PROGRAM PRG_03_Saw
VAR
	b_SRout: BOOL;	
	SR_saw: SR;
	R_TRIG_0: R_TRIG;
	R_TRIG_1: R_TRIG;
	R_TRIG_3: R_TRIG;
	R_TRIG_2: R_TRIG;
	R_TRIG_4: R_TRIG;
END_VAR
VAR // added by the converter: edge detectors and wires of the graphical bodies
    _w1 : BOOL;
END_VAR

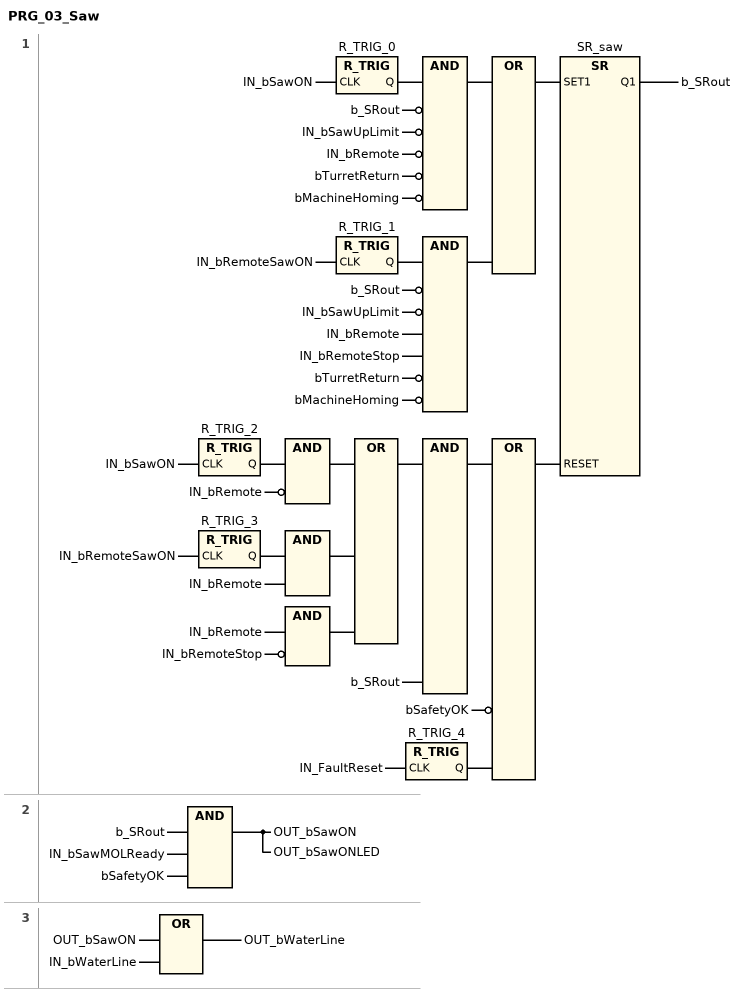
// NETWORK 1
R_TRIG_0(CLK := IN_bSawON); // R_TRIG
R_TRIG_1(CLK := IN_bRemoteSawON); // R_TRIG
R_TRIG_2(CLK := IN_bSawON); // R_TRIG
R_TRIG_3(CLK := IN_bRemoteSawON); // R_TRIG
R_TRIG_4(CLK := IN_FaultReset); // R_TRIG
SR_saw(SET1 := R_TRIG_0.Q AND NOT b_SRout AND NOT IN_bSawUpLimit AND NOT IN_bRemote AND NOT bTurretReturn AND NOT bMachineHoming OR R_TRIG_1.Q AND NOT b_SRout AND NOT IN_bSawUpLimit AND IN_bRemote AND IN_bRemoteStop AND NOT bTurretReturn AND NOT bMachineHoming, RESET := (R_TRIG_2.Q AND NOT IN_bRemote OR R_TRIG_3.Q AND IN_bRemote OR IN_bRemote AND NOT IN_bRemoteStop) AND b_SRout OR NOT bSafetyOK OR R_TRIG_4.Q); // SR
b_SRout := SR_saw.Q1;

// NETWORK 2
_w1 := b_SRout AND IN_bSawMOLReady AND bSafetyOK;
OUT_bSawON := _w1;
OUT_bSawONLED := _w1;

// NETWORK 3
OUT_bWaterLine := OUT_bSawON OR IN_bWaterLine;

END_PROGRAM

(* stored: Version 1.1.0.1, ProductVersion 3.1.4024.12
   POU PRG_03_Saw: Id {61e1e967-7bc0-48ef-8677-5ce5b6d3b95c}, SpecialFunc None *)
